TYPE ST_AxisReferenceFileConfig :
STRUCT
	Source : STRING(255);
	Target : STRING(80);
END_STRUCT
END_TYPE

(* stored: Version 1.1.0.1, ProductVersion 3.1.4026.18
   DUT ST_AxisReferenceFileConfig: Id {7f1821b8-9384-4455-9eb8-ed7083d28fb2} *)
